TYPE U_KRC_Output :
UNION
	aStdOut		AT %Q*		:ARRAY [0..3] OF DWORD;
	Control					:ST_KRC_Control;	
END_UNION
END_TYPE

(* stored: Version 1.1.0.1, ProductVersion 3.1.4024.10
   DUT U_KRC_Output: Id {840ff92b-13f7-4b50-9170-4952ef8224db} *)
